Omron CX-Programmer project NewProject (CX-Programmer 9.73)

# PLC NewPLC1: CJ2M CPU11

## Global symbols (name address type ; comment)
D0.00 BOOL  ; Eixo X
D100 CHANNEL  ; Paletes Completas
D1000.00 BOOL  ; Sensor_P
D1000.01 BOOL  ; Sensor_M
D1000.02 BOOL  ; Sensor_G
D1000.03 BOOL  ; TI_P
D1000.04 BOOL  ; TI_M
D1000.05 BOOL  ; TI_G
D1000.06 BOOL  ; TF_P
D1000.07 BOOL  ; TF_M
D1000.08 BOOL  ; TF_G
D1000.09 BOOL  ; START
D1000.10 BOOL  ; STOP
D1000.11 BOOL  ; SensorPI
D1000.12 BOOL  ; Pick_Enable
D1000.13 BOOL  ; SensorPF
D1000.14 BOOL  ; C Limit
D1001.00 BOOL  ; Sensor_Palete
D1001.01 BOOL  ; Manual
D1001.02 BOOL  ; Auto
D1001.03 BOOL  ; Emergencia
D1001.04 BOOL  ; RESET
D101 CHANNEL  ; Cx Pequenas
D102 CHANNEL  ; Cx Médias
D103 CHANNEL  ; Cx Grandes
D104 CHANNEL  ; Eixo X Pick&Place
D104.00 BOOL  ; SPX
D105 CHANNEL  ; Eixo Y Pick&Place
D105.00 BOOL  ; SPY
D106 CHANNEL  ; Eixo Z Pick&Place
D106.00 BOOL  ; SPZ
D1.00 BOOL  ; Eixo Y
D2000.00 BOOL  ; TI
D2000.01 BOOL  ; Frente
D2000.02 BOOL  ; Esquerda
D2000.03 BOOL  ; Direita
D2000.04 BOOL  ; T_M
D2000.05 BOOL  ; T_P
D2000.06 BOOL  ; T_G
D2000.12 BOOL  ; GRAB
D2000.13 BOOL  ; Start_Light
D2000.14 BOOL  ; Stop_Light
D2001.01 BOOL  ; Remove_PaleteM
D2001.02 BOOL  ; Remove_PaleteP
D2001.03 BOOL  ; Remove_PaleteFull
D2001.04 BOOL  ; Atras
D2001.05 BOOL  ; Reset_Light
D2001.06 BOOL  ; Remove_PaleteG
D2001.07 BOOL  ; T_Palete
D2001.08 BOOL  ; Palete_Spawn
D2001.09 BOOL  ; Palete_Receive
D2001.10 BOOL  ; 90_ROT
D200.00 BOOL  ; E0- Sistema desligado
D200.01 BOOL  ; E1 - Sistema ligado
D200.02 BOOL  ; E2 - Decisão
D200.03 BOOL  ; E3 - Mover caixa pequena
D200.04 BOOL  ; E4 - Mover caixa média
D200.05 BOOL  ; E5 - Mover caixa grande
D200.06 BOOL  ; E6 - Palete Pronta
D200.07 BOOL  ; E7 - Braço elevado
D200.08 BOOL  ; E8 - X,Y Cx Pequena
D200.09 BOOL  ; E9 - X,Y Cx Média
D200.10 BOOL  ; E10 - X,Y Cx Grande
D200.11 BOOL  ; E11 - Pegar Cx Pequena
D200.12 BOOL  ; E12 - Pegar Cx Média
D200.13 BOOL  ; E13 - Pegar Cx Grande
D200.14 BOOL  ; E14 - Caixa recolhida
D200.15 BOOL  ; E15 - Palete Cx Pequena
D201.00 BOOL  ; E16 - Palete Cx Pequena x2
D201.01 BOOL  ; E17 - Palete Cx Média
D201.02 BOOL  ; E18 - Palete Cx Grande
D201.03 BOOL  ; E19.0 - Drop Caixa pequena
D201.04 BOOL  ; E20 - Drop Caixa grande
D201.05 BOOL  ; E21 - Caixa colocada
D201.06 BOOL  ; E22 - Palete Pronta
D201.07 BOOL  ; E23 - Recolher Palete
D201.08 BOOL  ; E19.1 - Drop Caixa pequena x2
D201.09 BOOL  ; E19.2 - Drop Caixa média
D2.00 BOOL  ; Eixo Z
D300.00 BOOL  ; ON
D300.01 BOOL  ; MP
D300.02 BOOL  ; MM
D300.03 BOOL  ; MG
D300.04 BOOL  ; PickInicio
D300.05 BOOL  ; Remove_PaleteG ON
D300.07 BOOL  ; PickPequena
D300.08 BOOL  ; PickMedia
D300.09 BOOL  ; PickGrande
D300.10 BOOL  ; Emergencia_ON
D300.11 BOOL  ; Auto_ON
D302.00 BOOL  ; Y>=3.69
D302.01 BOOL  ; Y<=371
D302.02 BOOL  ; Z>=7.69
D302.03 BOOL  ; Z<=7.71
D302.04 BOOL  ; Z>=5.29
D302.05 BOOL  ; Z<=5.31
D302.06 BOOL  ; Y>=2.59
D302.07 BOOL  ; Z<=2.61
D302.08 BOOL  ; Y>=1.29
D302.09 BOOL  ; Y<=1.31
D303.00 BOOL  ; Z=0
D303.01 BOOL  ; Y=3.7
D303.02 BOOL  ; Y=10
D303.03 BOOL  ; Z=7.7
D303.04 BOOL  ; Z=5.3
D303.05 BOOL  ; Y=2.6
D303.06 BOOL  ; Y=1.3
D303.07 BOOL  ; Y=0
D303.08 BOOL  ; Z=10
D304.00 BOOL  ; Move Cx_Pequena
D304.01 BOOL  ; Move Cx_Media
D304.02 BOOL  ; Move Cx_Grande
D304.03 BOOL  ; Pick Cx_Pequena
D304.04 BOOL  ; Drop Cx_Pequena1
D304.05 BOOL  ; Drop Cx_Pequena2
D304.06 BOOL  ; Pick Cx_Media
D304.07 BOOL  ; Drop Cx_Media
D304.08 BOOL  ; Pick Cx_Grande
D304.09 BOOL  ; Drop Cx_Grande
D304.10 BOOL  ; Move_Decisao
D304.11 BOOL  ; Tapete_Final
D304.12 BOOL  ; System_ON
D304.13 BOOL  ; Decisao_Ready
D304.14 BOOL  ; Control_Emergencia
D304.15 BOOL  ; Control_Auto
T0002 BOOL  ; Timer_MoveDecisao

## Program NewProgram1 (cyclic task 0)

### Section ACOES

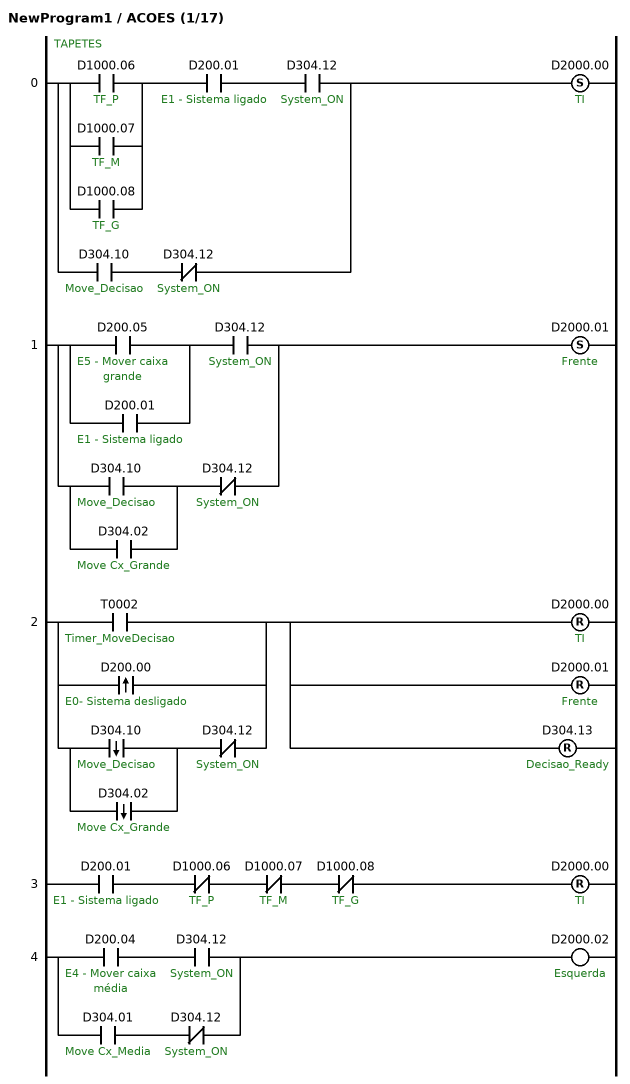
; rung 0: TAPETES
LD D1000.06  ; TF_P
OR D1000.07  ; TF_M
OR D1000.08  ; TF_G
AND D200.01  ; E1 - Sistema ligado
AND D304.12  ; System_ON
LD D304.10  ; Move_Decisao
ANDNOT D304.12  ; System_ON
ORLD
SET D2000.00  ; TI
; rung 1
LD D200.05  ; E5 - Mover caixa grande
OR D200.01  ; E1 - Sistema ligado
AND D304.12  ; System_ON
LD D304.10  ; Move_Decisao
OR D304.02  ; Move Cx_Grande
ANDNOT D304.12  ; System_ON
ORLD
SET D2000.01  ; Frente
; rung 2
LD T0002  ; Timer_MoveDecisao
@OR D200.00  ; E0- Sistema desligado
%LD D304.10  ; Move_Decisao
%OR D304.02  ; Move Cx_Grande
ANDNOT D304.12  ; System_ON
ORLD
RSET D2000.00  ; TI
RSET D2000.01  ; Frente
RSET D304.13  ; Decisao_Ready
; rung 3
LD D200.01  ; E1 - Sistema ligado
ANDNOT D1000.06  ; TF_P
ANDNOT D1000.07  ; TF_M
ANDNOT D1000.08  ; TF_G
RSET D2000.00  ; TI
; rung 4
LD D200.04  ; E4 - Mover caixa média
AND D304.12  ; System_ON
LD D304.01  ; Move Cx_Media
ANDNOT D304.12  ; System_ON
ORLD
OUT D2000.02  ; Esquerda

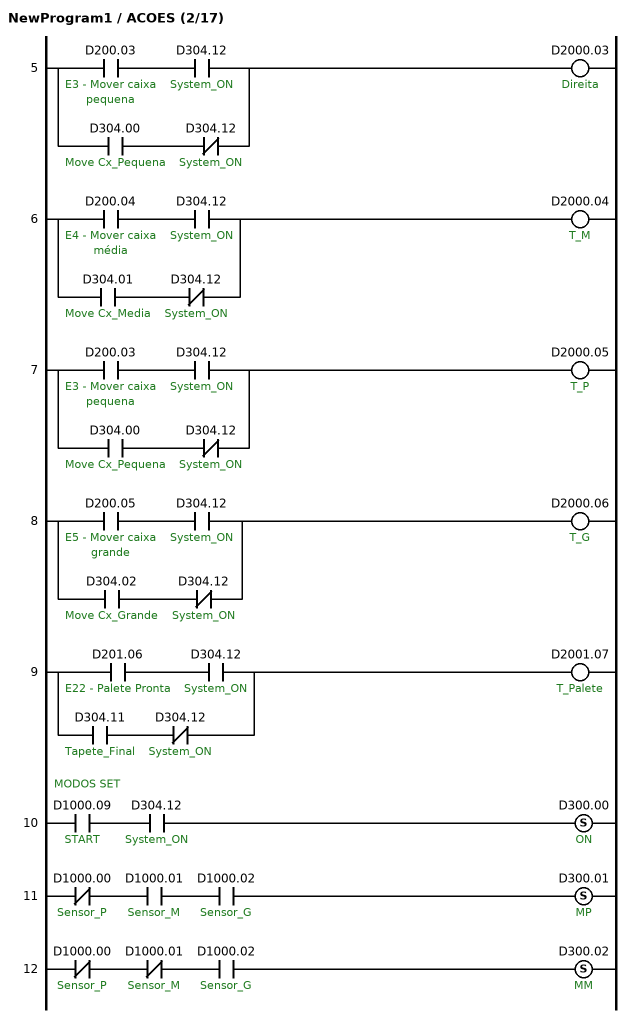
; rung 5
LD D200.03  ; E3 - Mover caixa pequena
AND D304.12  ; System_ON
LD D304.00  ; Move Cx_Pequena
ANDNOT D304.12  ; System_ON
ORLD
OUT D2000.03  ; Direita
; rung 6
LD D200.04  ; E4 - Mover caixa média
AND D304.12  ; System_ON
LD D304.01  ; Move Cx_Media
ANDNOT D304.12  ; System_ON
ORLD
OUT D2000.04  ; T_M
; rung 7
LD D200.03  ; E3 - Mover caixa pequena
AND D304.12  ; System_ON
LD D304.00  ; Move Cx_Pequena
ANDNOT D304.12  ; System_ON
ORLD
OUT D2000.05  ; T_P
; rung 8
LD D200.05  ; E5 - Mover caixa grande
AND D304.12  ; System_ON
LD D304.02  ; Move Cx_Grande
ANDNOT D304.12  ; System_ON
ORLD
OUT D2000.06  ; T_G
; rung 9
LD D201.06  ; E22 - Palete Pronta
AND D304.12  ; System_ON
LD D304.11  ; Tapete_Final
ANDNOT D304.12  ; System_ON
ORLD
OUT D2001.07  ; T_Palete
; rung 10: MODOS SET
LD D1000.09  ; START
AND D304.12  ; System_ON
SET D300.00  ; ON
; rung 11
LDNOT D1000.00  ; Sensor_P
AND D1000.01  ; Sensor_M
AND D1000.02  ; Sensor_G
SET D300.01  ; MP
; rung 12
LDNOT D1000.00  ; Sensor_P
ANDNOT D1000.01  ; Sensor_M
AND D1000.02  ; Sensor_G
SET D300.02  ; MM

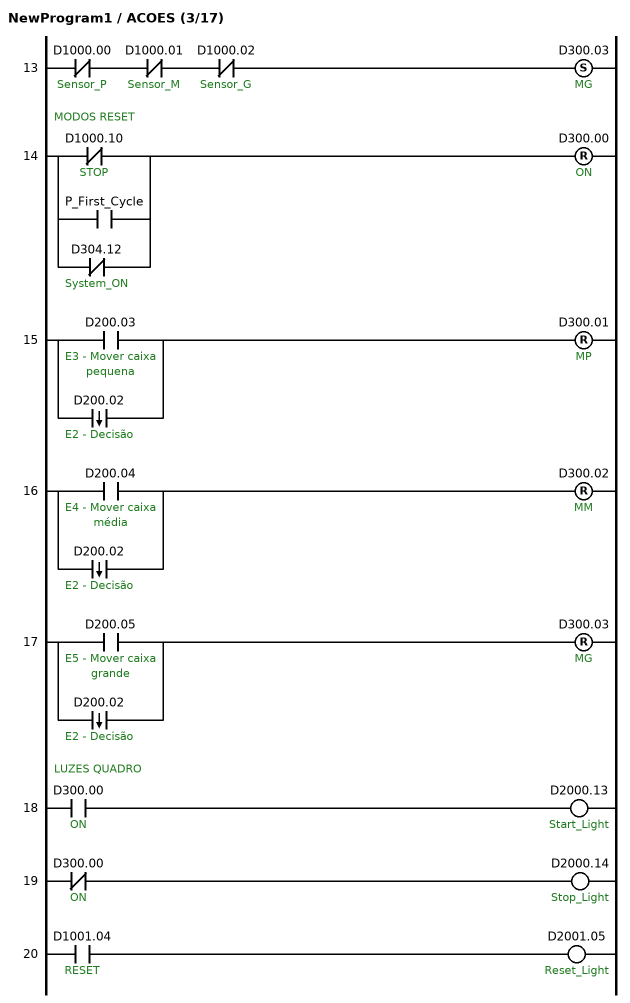
; rung 13
LDNOT D1000.00  ; Sensor_P
ANDNOT D1000.01  ; Sensor_M
ANDNOT D1000.02  ; Sensor_G
SET D300.03  ; MG
; rung 14: MODOS RESET
LDNOT D1000.10  ; STOP
OR P_First_Cycle
ORNOT D304.12  ; System_ON
RSET D300.00  ; ON
; rung 15
LD D200.03  ; E3 - Mover caixa pequena
%OR D200.02  ; E2 - Decisão
RSET D300.01  ; MP
; rung 16
LD D200.04  ; E4 - Mover caixa média
%OR D200.02  ; E2 - Decisão
RSET D300.02  ; MM
; rung 17
LD D200.05  ; E5 - Mover caixa grande
%OR D200.02  ; E2 - Decisão
RSET D300.03  ; MG
; rung 18: LUZES QUADRO
LD D300.00  ; ON
OUT D2000.13  ; Start_Light
; rung 19
LDNOT D300.00  ; ON
OUT D2000.14  ; Stop_Light
; rung 20
LD D1001.04  ; RESET
OUT D2001.05  ; Reset_Light

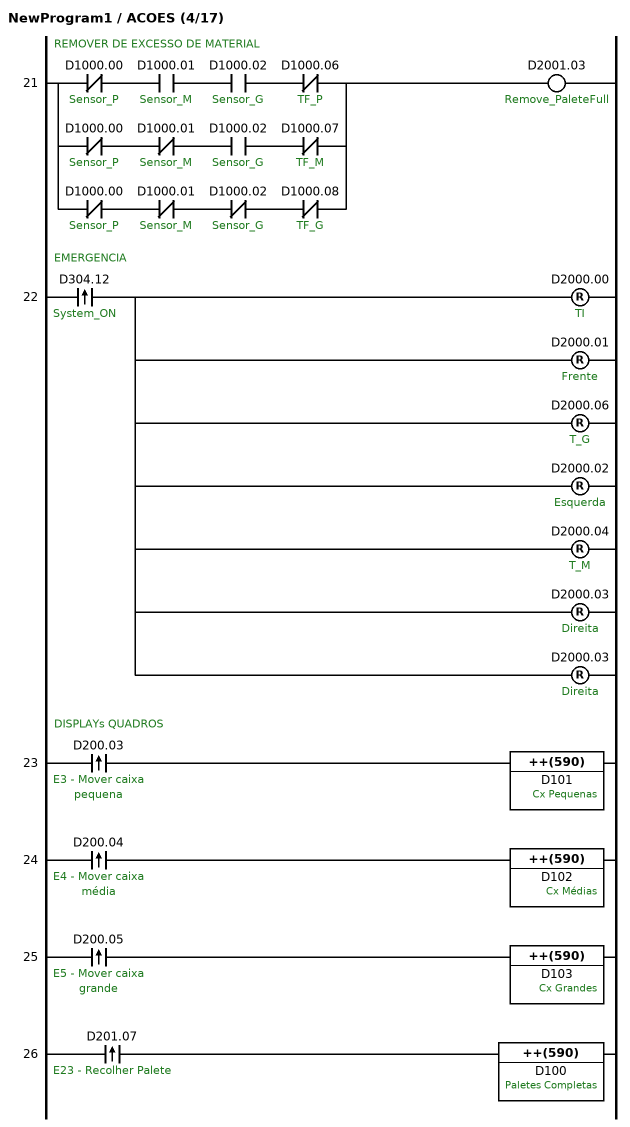
; rung 21: REMOVER DE EXCESSO DE MATERIAL
LDNOT D1000.00  ; Sensor_P
AND D1000.01  ; Sensor_M
AND D1000.02  ; Sensor_G
ANDNOT D1000.06  ; TF_P
LDNOT D1000.00  ; Sensor_P
ANDNOT D1000.01  ; Sensor_M
AND D1000.02  ; Sensor_G
ANDNOT D1000.07  ; TF_M
ORLD
LDNOT D1000.00  ; Sensor_P
ANDNOT D1000.01  ; Sensor_M
ANDNOT D1000.02  ; Sensor_G
ANDNOT D1000.08  ; TF_G
ORLD
OUT D2001.03  ; Remove_PaleteFull
; rung 22: EMERGENCIA
@LD D304.12  ; System_ON
RSET D2000.00  ; TI
RSET D2000.01  ; Frente
RSET D2000.06  ; T_G
RSET D2000.02  ; Esquerda
RSET D2000.04  ; T_M
RSET D2000.03  ; Direita
RSET D2000.03  ; Direita
; rung 23: DISPLAYs QUADROS
@LD D200.03  ; E3 - Mover caixa pequena
++(590) D101  ; Cx Pequenas
; rung 24
@LD D200.04  ; E4 - Mover caixa média
++(590) D102  ; Cx Médias
; rung 25
@LD D200.05  ; E5 - Mover caixa grande
++(590) D103  ; Cx Grandes
; rung 26
@LD D201.07  ; E23 - Recolher Palete
++(590) D100  ; Paletes Completas

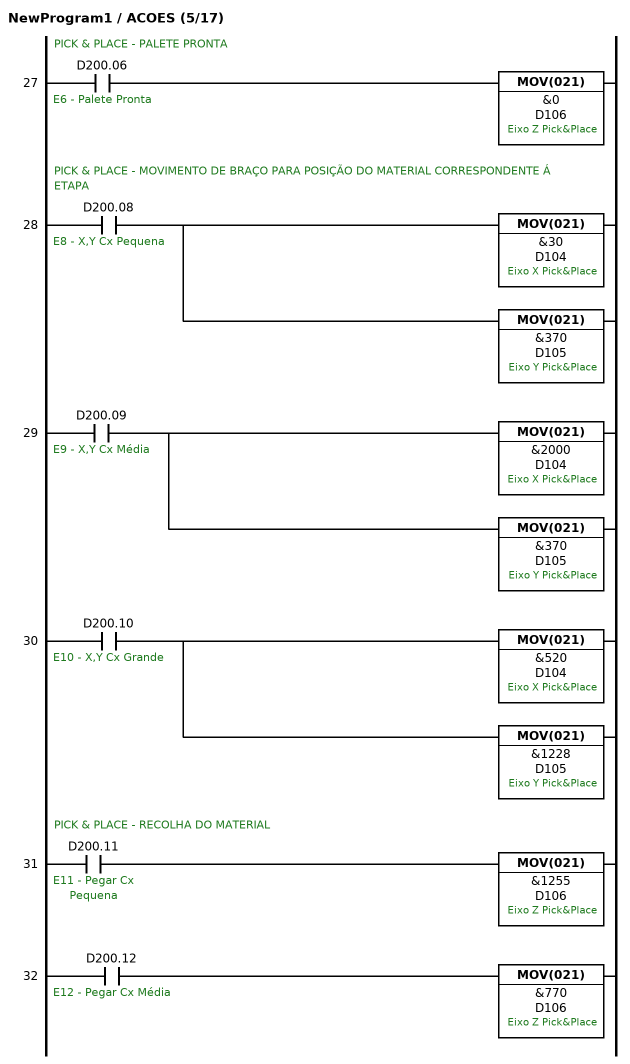
; rung 27: PICK & PLACE - PALETE PRONTA
LD D200.06  ; E6 - Palete Pronta
MOV(021) &0 D106  ; Eixo Z Pick&Place
; rung 28: PICK & PLACE - MOVIMENTO DE BRAÇO PARA POSIÇÃO DO MATERIAL CORRESPONDENTE Á ETAPA
LD D200.08  ; E8 - X,Y Cx Pequena
MOV(021) &30 D104  ; Eixo X Pick&Place
MOV(021) &370 D105  ; Eixo Y Pick&Place
; rung 29
LD D200.09  ; E9 - X,Y Cx Média
MOV(021) &2000 D104  ; Eixo X Pick&Place
MOV(021) &370 D105  ; Eixo Y Pick&Place
; rung 30
LD D200.10  ; E10 - X,Y Cx Grande
MOV(021) &520 D104  ; Eixo X Pick&Place
MOV(021) &1228 D105  ; Eixo Y Pick&Place
; rung 31: PICK & PLACE - RECOLHA DO MATERIAL
LD D200.11  ; E11 - Pegar Cx Pequena
MOV(021) &1255 D106  ; Eixo Z Pick&Place
; rung 32
LD D200.12  ; E12 - Pegar Cx Média
MOV(021) &770 D106  ; Eixo Z Pick&Place

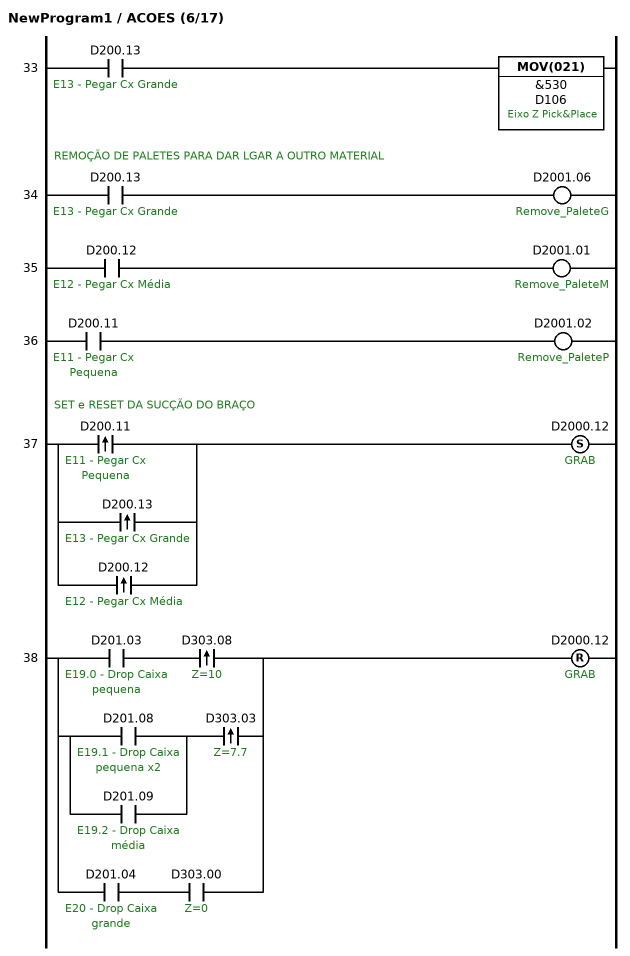
; rung 33
LD D200.13  ; E13 - Pegar Cx Grande
MOV(021) &530 D106  ; Eixo Z Pick&Place
; rung 34: REMOÇÃO DE PALETES PARA DAR LGAR A OUTRO MATERIAL
LD D200.13  ; E13 - Pegar Cx Grande
OUT D2001.06  ; Remove_PaleteG
; rung 35
LD D200.12  ; E12 - Pegar Cx Média
OUT D2001.01  ; Remove_PaleteM
; rung 36
LD D200.11  ; E11 - Pegar Cx Pequena
OUT D2001.02  ; Remove_PaleteP
; rung 37: SET e RESET DA SUCÇÃO DO BRAÇO
@LD D200.11  ; E11 - Pegar Cx Pequena
@OR D200.13  ; E13 - Pegar Cx Grande
@OR D200.12  ; E12 - Pegar Cx Média
SET D2000.12  ; GRAB
; rung 38
LD D201.03  ; E19.0 - Drop Caixa pequena
@AND D303.08  ; Z=10
LD D201.08  ; E19.1 - Drop Caixa pequena x2
OR D201.09  ; E19.2 - Drop Caixa média
@AND D303.03  ; Z=7.7
ORLD
LD D201.04  ; E20 - Drop Caixa grande
AND D303.00  ; Z=0
ORLD
RSET D2000.12  ; GRAB

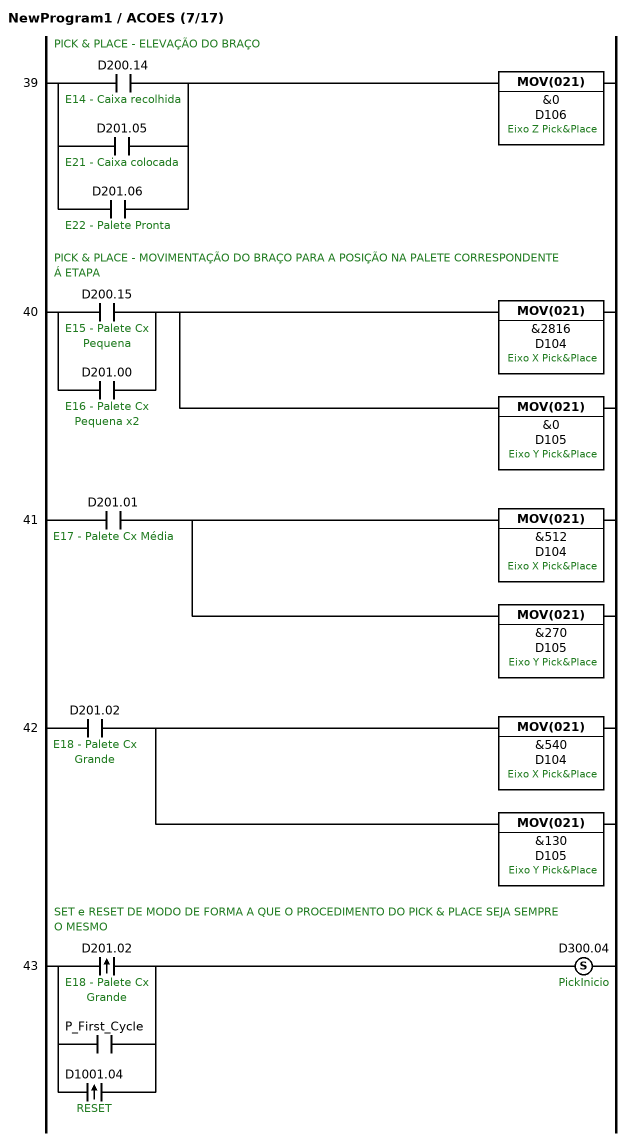
; rung 39: PICK & PLACE - ELEVAÇÃO DO BRAÇO
LD D200.14  ; E14 - Caixa recolhida
OR D201.05  ; E21 - Caixa colocada
OR D201.06  ; E22 - Palete Pronta
MOV(021) &0 D106  ; Eixo Z Pick&Place
; rung 40: PICK & PLACE - MOVIMENTAÇÃO DO BRAÇO PARA A POSIÇÃO NA PALETE CORRESPONDENTE Á ETAPA
LD D200.15  ; E15 - Palete Cx Pequena
OR D201.00  ; E16 - Palete Cx Pequena x2
MOV(021) &2816 D104  ; Eixo X Pick&Place
MOV(021) &0 D105  ; Eixo Y Pick&Place
; rung 41
LD D201.01  ; E17 - Palete Cx Média
MOV(021) &512 D104  ; Eixo X Pick&Place
MOV(021) &270 D105  ; Eixo Y Pick&Place
; rung 42
LD D201.02  ; E18 - Palete Cx Grande
MOV(021) &540 D104  ; Eixo X Pick&Place
MOV(021) &130 D105  ; Eixo Y Pick&Place
; rung 43: SET e RESET DE MODO DE FORMA A QUE O PROCEDIMENTO DO PICK & PLACE SEJA SEMPRE O MESMO
@LD D201.02  ; E18 - Palete Cx Grande
OR P_First_Cycle
@OR D1001.04  ; RESET
SET D300.04  ; PickInicio

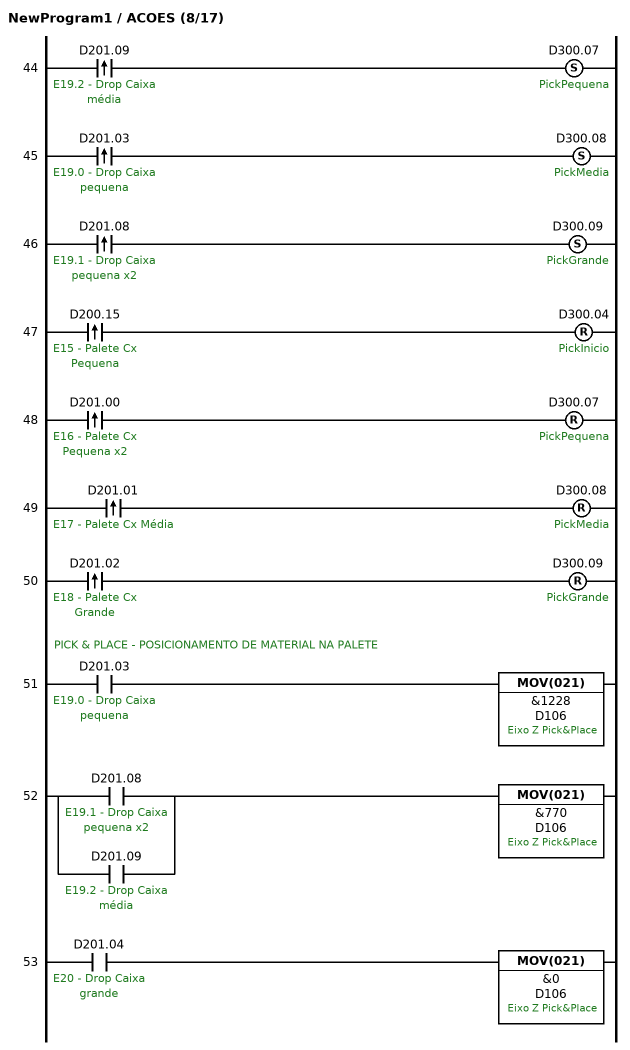
; rung 44
@LD D201.09  ; E19.2 - Drop Caixa média
SET D300.07  ; PickPequena
; rung 45
@LD D201.03  ; E19.0 - Drop Caixa pequena
SET D300.08  ; PickMedia
; rung 46
@LD D201.08  ; E19.1 - Drop Caixa pequena x2
SET D300.09  ; PickGrande
; rung 47
@LD D200.15  ; E15 - Palete Cx Pequena
RSET D300.04  ; PickInicio
; rung 48
@LD D201.00  ; E16 - Palete Cx Pequena x2
RSET D300.07  ; PickPequena
; rung 49
@LD D201.01  ; E17 - Palete Cx Média
RSET D300.08  ; PickMedia
; rung 50
@LD D201.02  ; E18 - Palete Cx Grande
RSET D300.09  ; PickGrande
; rung 51: PICK & PLACE - POSICIONAMENTO DE MATERIAL NA PALETE
LD D201.03  ; E19.0 - Drop Caixa pequena
MOV(021) &1228 D106  ; Eixo Z Pick&Place
; rung 52
LD D201.08  ; E19.1 - Drop Caixa pequena x2
OR D201.09  ; E19.2 - Drop Caixa média
MOV(021) &770 D106  ; Eixo Z Pick&Place
; rung 53
LD D201.04  ; E20 - Drop Caixa grande
MOV(021) &0 D106  ; Eixo Z Pick&Place

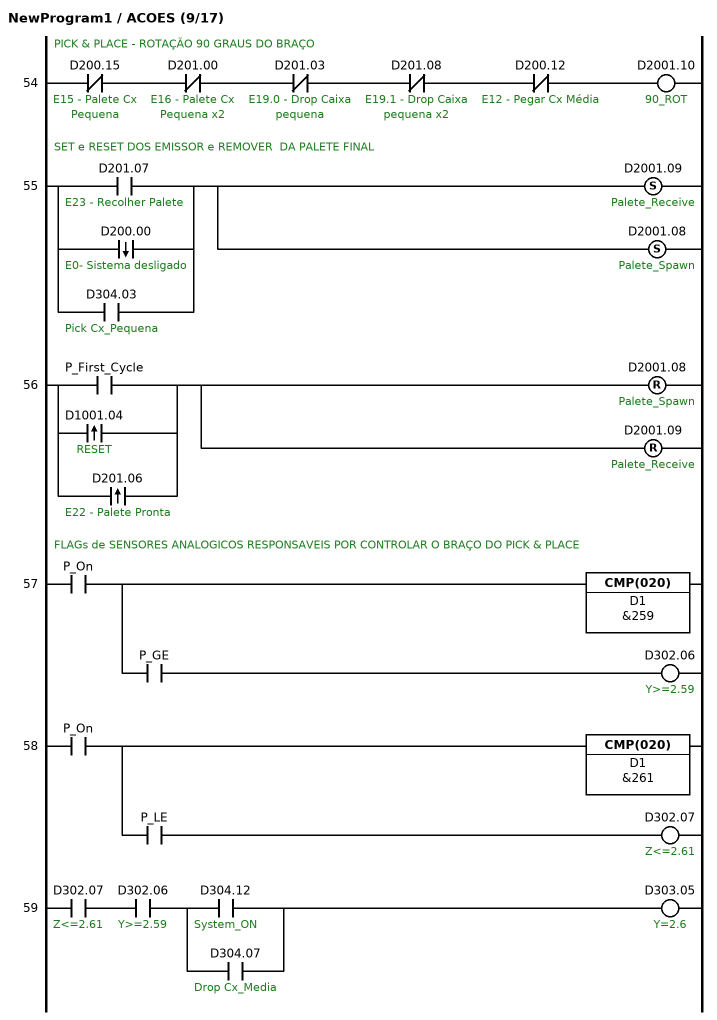
; rung 54: PICK & PLACE - ROTAÇÃO 90 GRAUS DO BRAÇO
LDNOT D200.15  ; E15 - Palete Cx Pequena
ANDNOT D201.00  ; E16 - Palete Cx Pequena x2
ANDNOT D201.03  ; E19.0 - Drop Caixa pequena
ANDNOT D201.08  ; E19.1 - Drop Caixa pequena x2
ANDNOT D200.12  ; E12 - Pegar Cx Média
OUT D2001.10  ; 90_ROT
; rung 55: SET e RESET DOS EMISSOR e REMOVER  DA PALETE FINAL
LD D201.07  ; E23 - Recolher Palete
%OR D200.00  ; E0- Sistema desligado
OR D304.03  ; Pick Cx_Pequena
SET D2001.09  ; Palete_Receive
SET D2001.08  ; Palete_Spawn
; rung 56
LD P_First_Cycle
@OR D1001.04  ; RESET
@OR D201.06  ; E22 - Palete Pronta
RSET D2001.08  ; Palete_Spawn
RSET D2001.09  ; Palete_Receive
; rung 57: FLAGs de SENSORES ANALOGICOS RESPONSAVEIS POR CONTROLAR O BRAÇO DO PICK & PLACE
LD P_On
CMP(020) D1 &259
AND P_GE
OUT D302.06  ; Y>=2.59
; rung 58
LD P_On
CMP(020) D1 &261
AND P_LE
OUT D302.07  ; Z<=2.61
; rung 59
LD D302.07  ; Z<=2.61
AND D302.06  ; Y>=2.59
LD D304.12  ; System_ON
OR D304.07  ; Drop Cx_Media
ANDLD
OUT D303.05  ; Y=2.6

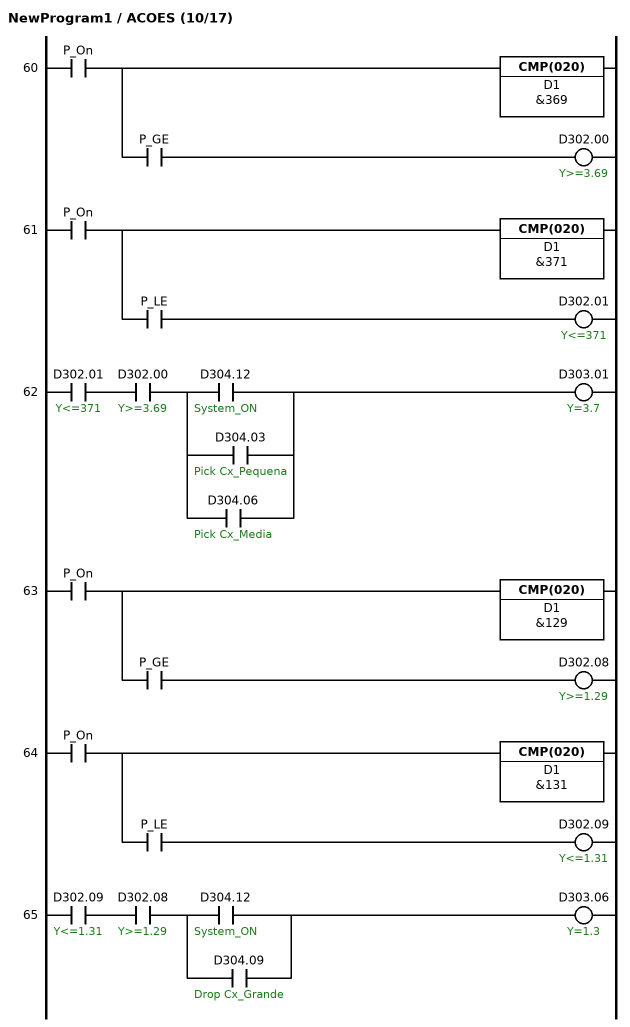
; rung 60
LD P_On
CMP(020) D1 &369
AND P_GE
OUT D302.00  ; Y>=3.69
; rung 61
LD P_On
CMP(020) D1 &371
AND P_LE
OUT D302.01  ; Y<=371
; rung 62
LD D302.01  ; Y<=371
AND D302.00  ; Y>=3.69
LD D304.12  ; System_ON
OR D304.03  ; Pick Cx_Pequena
OR D304.06  ; Pick Cx_Media
ANDLD
OUT D303.01  ; Y=3.7
; rung 63
LD P_On
CMP(020) D1 &129
AND P_GE
OUT D302.08  ; Y>=1.29
; rung 64
LD P_On
CMP(020) D1 &131
AND P_LE
OUT D302.09  ; Y<=1.31
; rung 65
LD D302.09  ; Y<=1.31
AND D302.08  ; Y>=1.29
LD D304.12  ; System_ON
OR D304.09  ; Drop Cx_Grande
ANDLD
OUT D303.06  ; Y=1.3

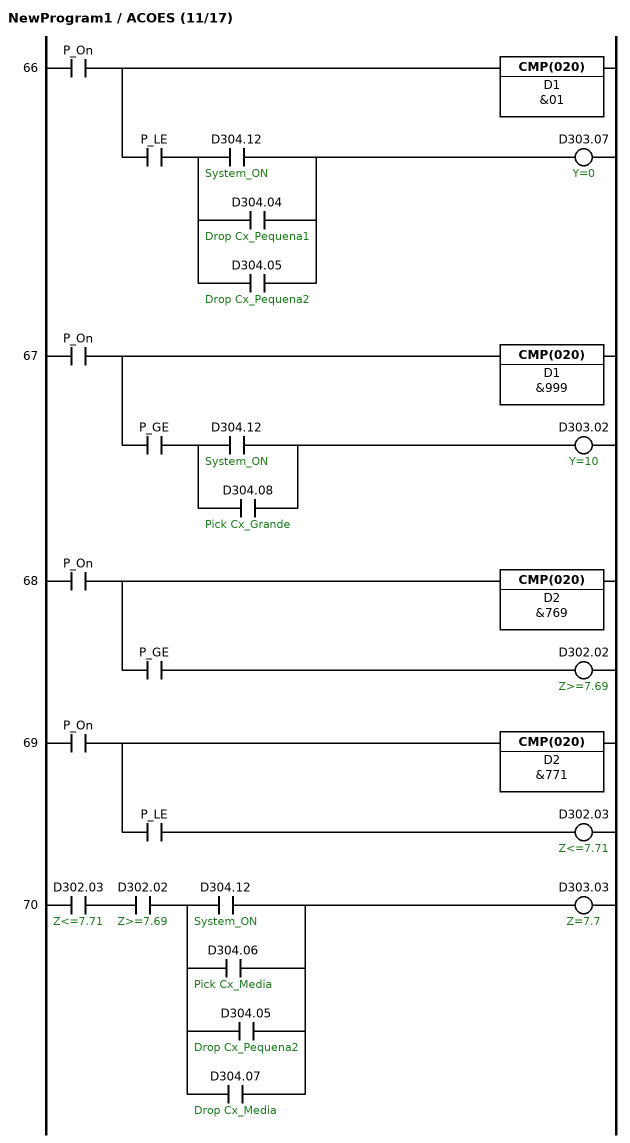
; rung 66
LD P_On
CMP(020) D1 &01
AND P_LE
LD D304.12  ; System_ON
OR D304.04  ; Drop Cx_Pequena1
OR D304.05  ; Drop Cx_Pequena2
ANDLD
OUT D303.07  ; Y=0
; rung 67
LD P_On
CMP(020) D1 &999
AND P_GE
LD D304.12  ; System_ON
OR D304.08  ; Pick Cx_Grande
ANDLD
OUT D303.02  ; Y=10
; rung 68
LD P_On
CMP(020) D2 &769
AND P_GE
OUT D302.02  ; Z>=7.69
; rung 69
LD P_On
CMP(020) D2 &771
AND P_LE
OUT D302.03  ; Z<=7.71
; rung 70
LD D302.03  ; Z<=7.71
AND D302.02  ; Z>=7.69
LD D304.12  ; System_ON
OR D304.06  ; Pick Cx_Media
OR D304.05  ; Drop Cx_Pequena2
OR D304.07  ; Drop Cx_Media
ANDLD
OUT D303.03  ; Z=7.7

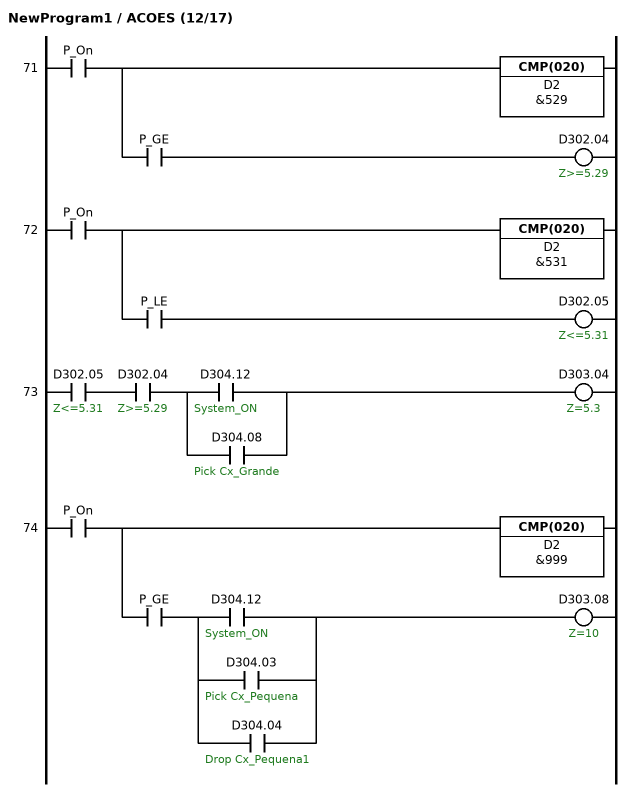
; rung 71
LD P_On
CMP(020) D2 &529
AND P_GE
OUT D302.04  ; Z>=5.29
; rung 72
LD P_On
CMP(020) D2 &531
AND P_LE
OUT D302.05  ; Z<=5.31
; rung 73
LD D302.05  ; Z<=5.31
AND D302.04  ; Z>=5.29
LD D304.12  ; System_ON
OR D304.08  ; Pick Cx_Grande
ANDLD
OUT D303.04  ; Z=5.3
; rung 74
LD P_On
CMP(020) D2 &999
AND P_GE
LD D304.12  ; System_ON
OR D304.03  ; Pick Cx_Pequena
OR D304.04  ; Drop Cx_Pequena1
ANDLD
OUT D303.08  ; Z=10

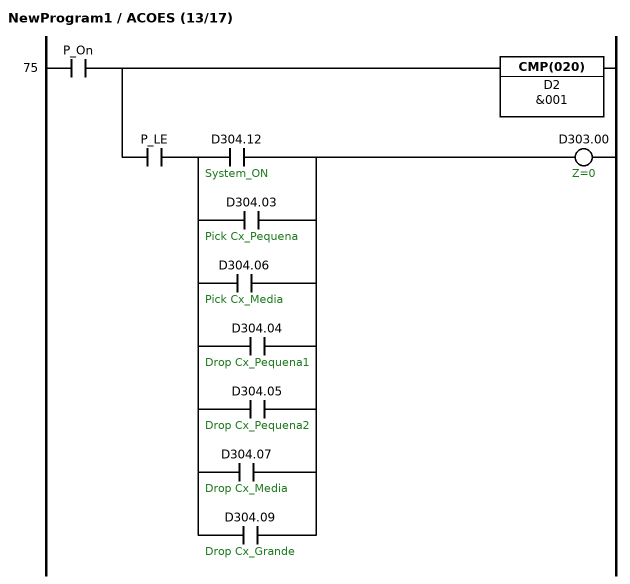
; rung 75
LD P_On
CMP(020) D2 &001
AND P_LE
LD D304.12  ; System_ON
OR D304.03  ; Pick Cx_Pequena
OR D304.06  ; Pick Cx_Media
OR D304.04  ; Drop Cx_Pequena1
OR D304.05  ; Drop Cx_Pequena2
OR D304.07  ; Drop Cx_Media
OR D304.09  ; Drop Cx_Grande
ANDLD
OUT D303.00  ; Z=0

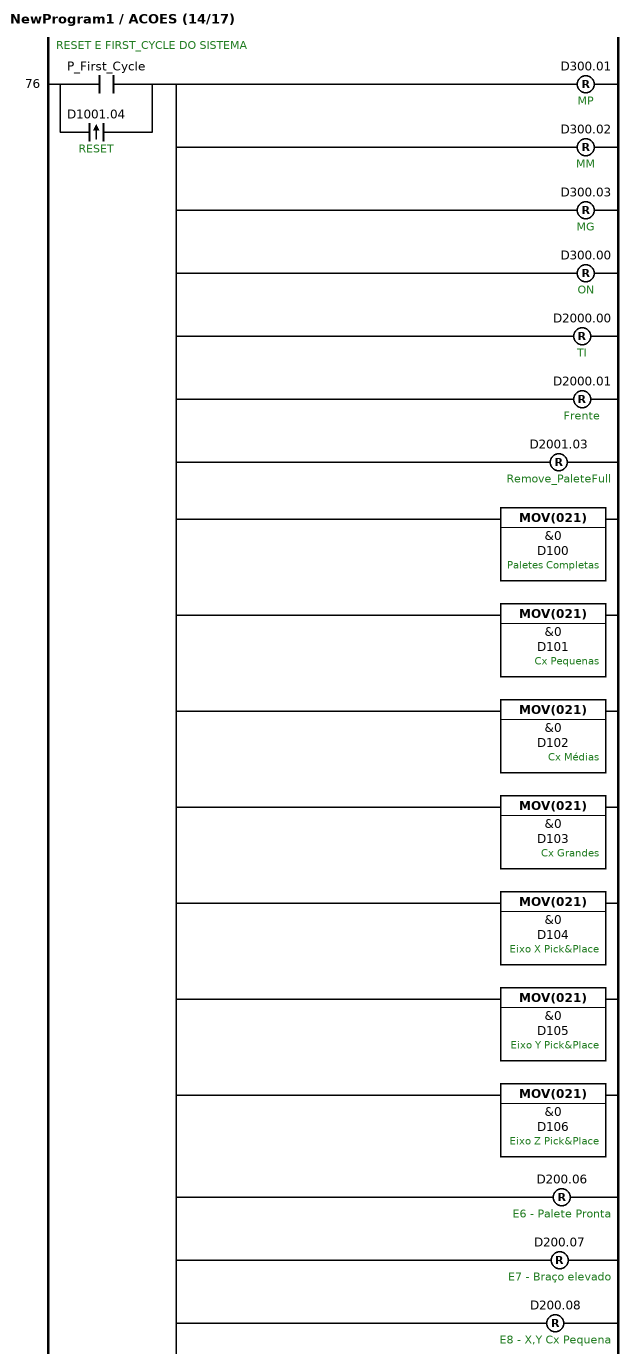

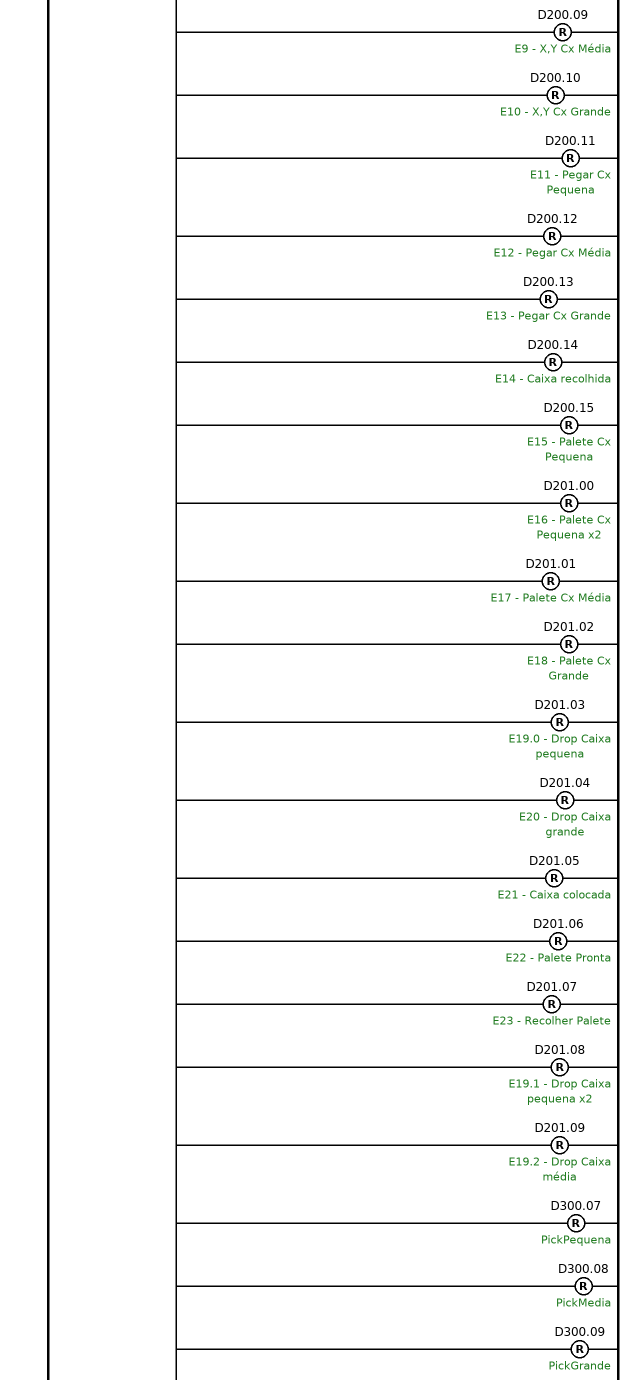

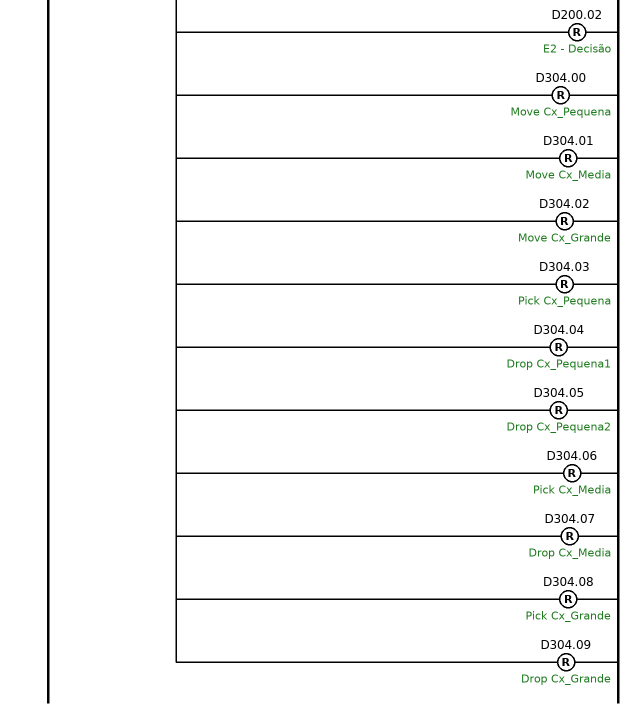
; rung 76: RESET E FIRST_CYCLE DO SISTEMA
LD P_First_Cycle
@OR D1001.04  ; RESET
RSET D300.01  ; MP
RSET D300.02  ; MM
RSET D300.03  ; MG
RSET D300.00  ; ON
RSET D2000.00  ; TI
RSET D2000.01  ; Frente
RSET D2001.03  ; Remove_PaleteFull
MOV(021) &0 D100  ; Paletes Completas
MOV(021) &0 D101  ; Cx Pequenas
MOV(021) &0 D102  ; Cx Médias
MOV(021) &0 D103  ; Cx Grandes
MOV(021) &0 D104  ; Eixo X Pick&Place
MOV(021) &0 D105  ; Eixo Y Pick&Place
MOV(021) &0 D106  ; Eixo Z Pick&Place
RSET D200.06  ; E6 - Palete Pronta
RSET D200.07  ; E7 - Braço elevado
RSET D200.08  ; E8 - X,Y Cx Pequena
RSET D200.09  ; E9 - X,Y Cx Média
RSET D200.10  ; E10 - X,Y Cx Grande
RSET D200.11  ; E11 - Pegar Cx Pequena
RSET D200.12  ; E12 - Pegar Cx Média
RSET D200.13  ; E13 - Pegar Cx Grande
RSET D200.14  ; E14 - Caixa recolhida
RSET D200.15  ; E15 - Palete Cx Pequena
RSET D201.00  ; E16 - Palete Cx Pequena x2
RSET D201.01  ; E17 - Palete Cx Média
RSET D201.02  ; E18 - Palete Cx Grande
RSET D201.03  ; E19.0 - Drop Caixa pequena
RSET D201.04  ; E20 - Drop Caixa grande
RSET D201.05  ; E21 - Caixa colocada
RSET D201.06  ; E22 - Palete Pronta
RSET D201.07  ; E23 - Recolher Palete
RSET D201.08  ; E19.1 - Drop Caixa pequena x2
RSET D201.09  ; E19.2 - Drop Caixa média
RSET D300.07  ; PickPequena
RSET D300.08  ; PickMedia
RSET D300.09  ; PickGrande
RSET D200.02  ; E2 - Decisão
RSET D304.00  ; Move Cx_Pequena
RSET D304.01  ; Move Cx_Media
RSET D304.02  ; Move Cx_Grande
RSET D304.03  ; Pick Cx_Pequena
RSET D304.04  ; Drop Cx_Pequena1
RSET D304.05  ; Drop Cx_Pequena2
RSET D304.06  ; Pick Cx_Media
RSET D304.07  ; Drop Cx_Media
RSET D304.08  ; Pick Cx_Grande
RSET D304.09  ; Drop Cx_Grande

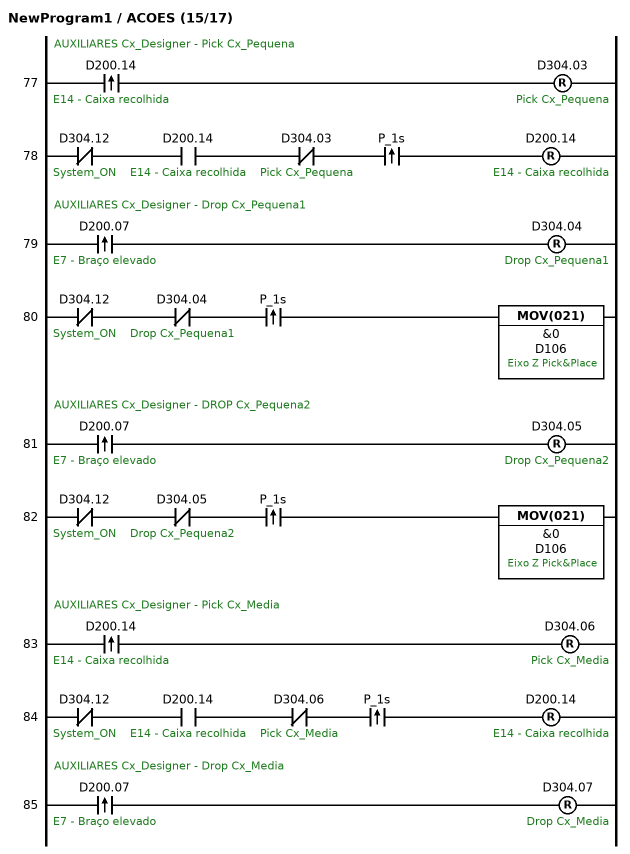
; rung 77: AUXILIARES Cx_Designer - Pick Cx_Pequena
@LD D200.14  ; E14 - Caixa recolhida
RSET D304.03  ; Pick Cx_Pequena
; rung 78
LDNOT D304.12  ; System_ON
AND D200.14  ; E14 - Caixa recolhida
ANDNOT D304.03  ; Pick Cx_Pequena
@AND P_1s
RSET D200.14  ; E14 - Caixa recolhida
; rung 79: AUXILIARES Cx_Designer - Drop Cx_Pequena1
@LD D200.07  ; E7 - Braço elevado
RSET D304.04  ; Drop Cx_Pequena1
; rung 80
LDNOT D304.12  ; System_ON
ANDNOT D304.04  ; Drop Cx_Pequena1
@AND P_1s
MOV(021) &0 D106  ; Eixo Z Pick&Place
; rung 81: AUXILIARES Cx_Designer - DROP Cx_Pequena2
@LD D200.07  ; E7 - Braço elevado
RSET D304.05  ; Drop Cx_Pequena2
; rung 82
LDNOT D304.12  ; System_ON
ANDNOT D304.05  ; Drop Cx_Pequena2
@AND P_1s
MOV(021) &0 D106  ; Eixo Z Pick&Place
; rung 83: AUXILIARES Cx_Designer - Pick Cx_Media
@LD D200.14  ; E14 - Caixa recolhida
RSET D304.06  ; Pick Cx_Media
; rung 84
LDNOT D304.12  ; System_ON
AND D200.14  ; E14 - Caixa recolhida
ANDNOT D304.06  ; Pick Cx_Media
@AND P_1s
RSET D200.14  ; E14 - Caixa recolhida
; rung 85: AUXILIARES Cx_Designer - Drop Cx_Media
@LD D200.07  ; E7 - Braço elevado
RSET D304.07  ; Drop Cx_Media

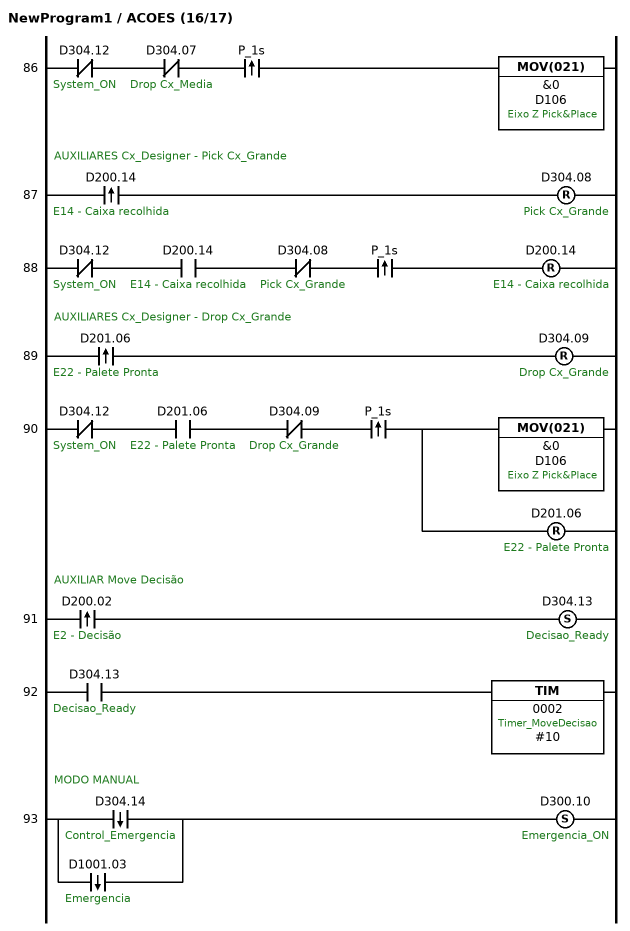
; rung 86
LDNOT D304.12  ; System_ON
ANDNOT D304.07  ; Drop Cx_Media
@AND P_1s
MOV(021) &0 D106  ; Eixo Z Pick&Place
; rung 87: AUXILIARES Cx_Designer - Pick Cx_Grande
@LD D200.14  ; E14 - Caixa recolhida
RSET D304.08  ; Pick Cx_Grande
; rung 88
LDNOT D304.12  ; System_ON
AND D200.14  ; E14 - Caixa recolhida
ANDNOT D304.08  ; Pick Cx_Grande
@AND P_1s
RSET D200.14  ; E14 - Caixa recolhida
; rung 89: AUXILIARES Cx_Designer - Drop Cx_Grande
@LD D201.06  ; E22 - Palete Pronta
RSET D304.09  ; Drop Cx_Grande
; rung 90
LDNOT D304.12  ; System_ON
AND D201.06  ; E22 - Palete Pronta
ANDNOT D304.09  ; Drop Cx_Grande
@AND P_1s
MOV(021) &0 D106  ; Eixo Z Pick&Place
RSET D201.06  ; E22 - Palete Pronta
; rung 91: AUXILIAR Move Decisão
@LD D200.02  ; E2 - Decisão
SET D304.13  ; Decisao_Ready
; rung 92
LD D304.13  ; Decisao_Ready
TIM 0002 #10  ; Timer_MoveDecisao
; rung 93: MODO MANUAL
%LD D304.14  ; Control_Emergencia
%OR D1001.03  ; Emergencia
SET D300.10  ; Emergencia_ON

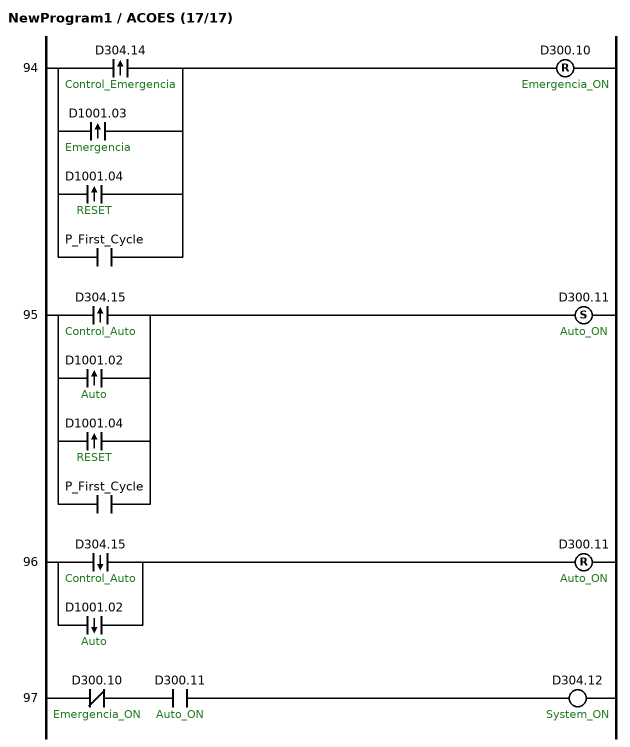
; rung 94
@LD D304.14  ; Control_Emergencia
@OR D1001.03  ; Emergencia
@OR D1001.04  ; RESET
OR P_First_Cycle
RSET D300.10  ; Emergencia_ON
; rung 95
@LD D304.15  ; Control_Auto
@OR D1001.02  ; Auto
@OR D1001.04  ; RESET
OR P_First_Cycle
SET D300.11  ; Auto_ON
; rung 96
%LD D304.15  ; Control_Auto
%OR D1001.02  ; Auto
RSET D300.11  ; Auto_ON
; rung 97
LDNOT D300.10  ; Emergencia_ON
AND D300.11  ; Auto_ON
OUT D304.12  ; System_ON

### Section ETAPAS

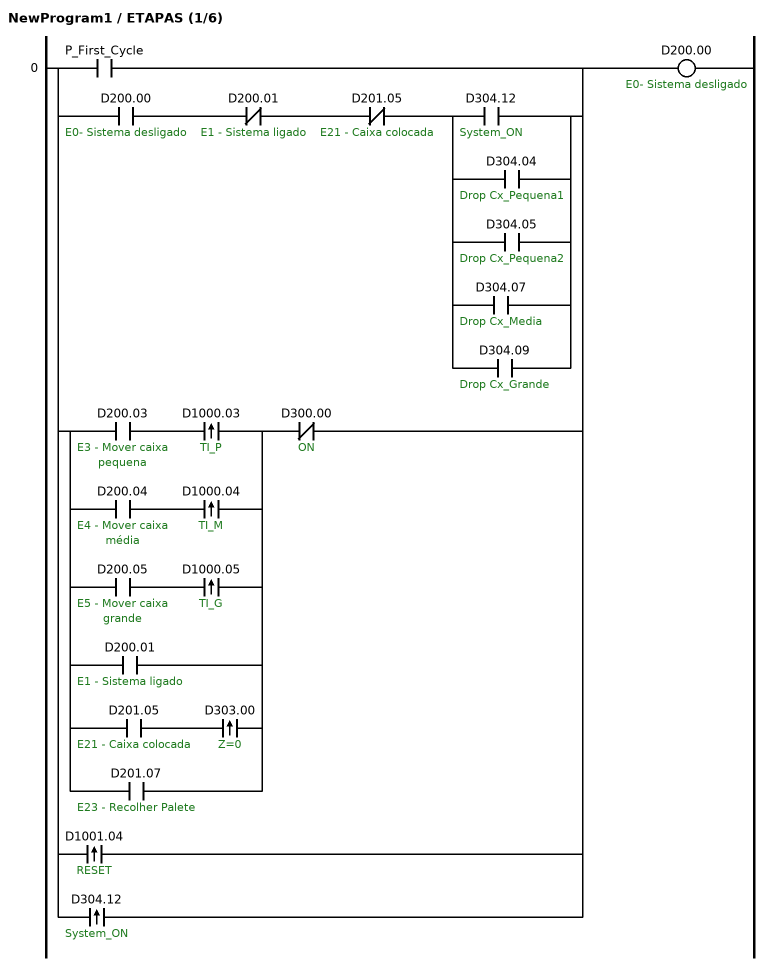
; rung 0
LD P_First_Cycle
LD D200.00  ; E0- Sistema desligado
ANDNOT D200.01  ; E1 - Sistema ligado
ANDNOT D201.05  ; E21 - Caixa colocada
LD D304.12  ; System_ON
OR D304.04  ; Drop Cx_Pequena1
OR D304.05  ; Drop Cx_Pequena2
OR D304.07  ; Drop Cx_Media
OR D304.09  ; Drop Cx_Grande
ANDLD
ORLD
LD D200.03  ; E3 - Mover caixa pequena
@AND D1000.03  ; TI_P
LD D200.04  ; E4 - Mover caixa média
@AND D1000.04  ; TI_M
ORLD
LD D200.05  ; E5 - Mover caixa grande
@AND D1000.05  ; TI_G
ORLD
OR D200.01  ; E1 - Sistema ligado
LD D201.05  ; E21 - Caixa colocada
@AND D303.00  ; Z=0
ORLD
OR D201.07  ; E23 - Recolher Palete
ANDNOT D300.00  ; ON
ORLD
@OR D1001.04  ; RESET
@OR D304.12  ; System_ON
OUT D200.00  ; E0- Sistema desligado

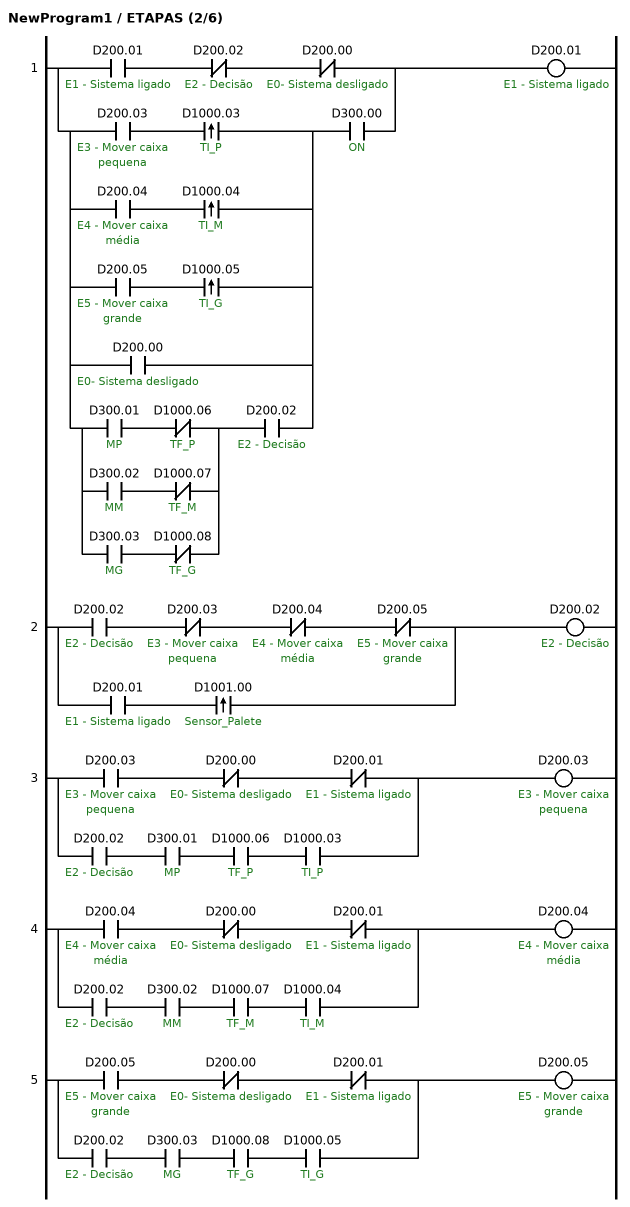
; rung 1
LD D200.01  ; E1 - Sistema ligado
ANDNOT D200.02  ; E2 - Decisão
ANDNOT D200.00  ; E0- Sistema desligado
LD D200.03  ; E3 - Mover caixa pequena
@AND D1000.03  ; TI_P
LD D200.04  ; E4 - Mover caixa média
@AND D1000.04  ; TI_M
ORLD
LD D200.05  ; E5 - Mover caixa grande
@AND D1000.05  ; TI_G
ORLD
OR D200.00  ; E0- Sistema desligado
LD D300.01  ; MP
ANDNOT D1000.06  ; TF_P
LD D300.02  ; MM
ANDNOT D1000.07  ; TF_M
ORLD
LD D300.03  ; MG
ANDNOT D1000.08  ; TF_G
ORLD
AND D200.02  ; E2 - Decisão
ORLD
AND D300.00  ; ON
ORLD
OUT D200.01  ; E1 - Sistema ligado
; rung 2
LD D200.02  ; E2 - Decisão
ANDNOT D200.03  ; E3 - Mover caixa pequena
ANDNOT D200.04  ; E4 - Mover caixa média
ANDNOT D200.05  ; E5 - Mover caixa grande
LD D200.01  ; E1 - Sistema ligado
@AND D1001.00  ; Sensor_Palete
ORLD
OUT D200.02  ; E2 - Decisão
; rung 3
LD D200.03  ; E3 - Mover caixa pequena
ANDNOT D200.00  ; E0- Sistema desligado
ANDNOT D200.01  ; E1 - Sistema ligado
LD D200.02  ; E2 - Decisão
AND D300.01  ; MP
AND D1000.06  ; TF_P
AND D1000.03  ; TI_P
ORLD
OUT D200.03  ; E3 - Mover caixa pequena
; rung 4
LD D200.04  ; E4 - Mover caixa média
ANDNOT D200.00  ; E0- Sistema desligado
ANDNOT D200.01  ; E1 - Sistema ligado
LD D200.02  ; E2 - Decisão
AND D300.02  ; MM
AND D1000.07  ; TF_M
AND D1000.04  ; TI_M
ORLD
OUT D200.04  ; E4 - Mover caixa média
; rung 5
LD D200.05  ; E5 - Mover caixa grande
ANDNOT D200.00  ; E0- Sistema desligado
ANDNOT D200.01  ; E1 - Sistema ligado
LD D200.02  ; E2 - Decisão
AND D300.03  ; MG
AND D1000.08  ; TF_G
AND D1000.05  ; TI_G
ORLD
OUT D200.05  ; E5 - Mover caixa grande

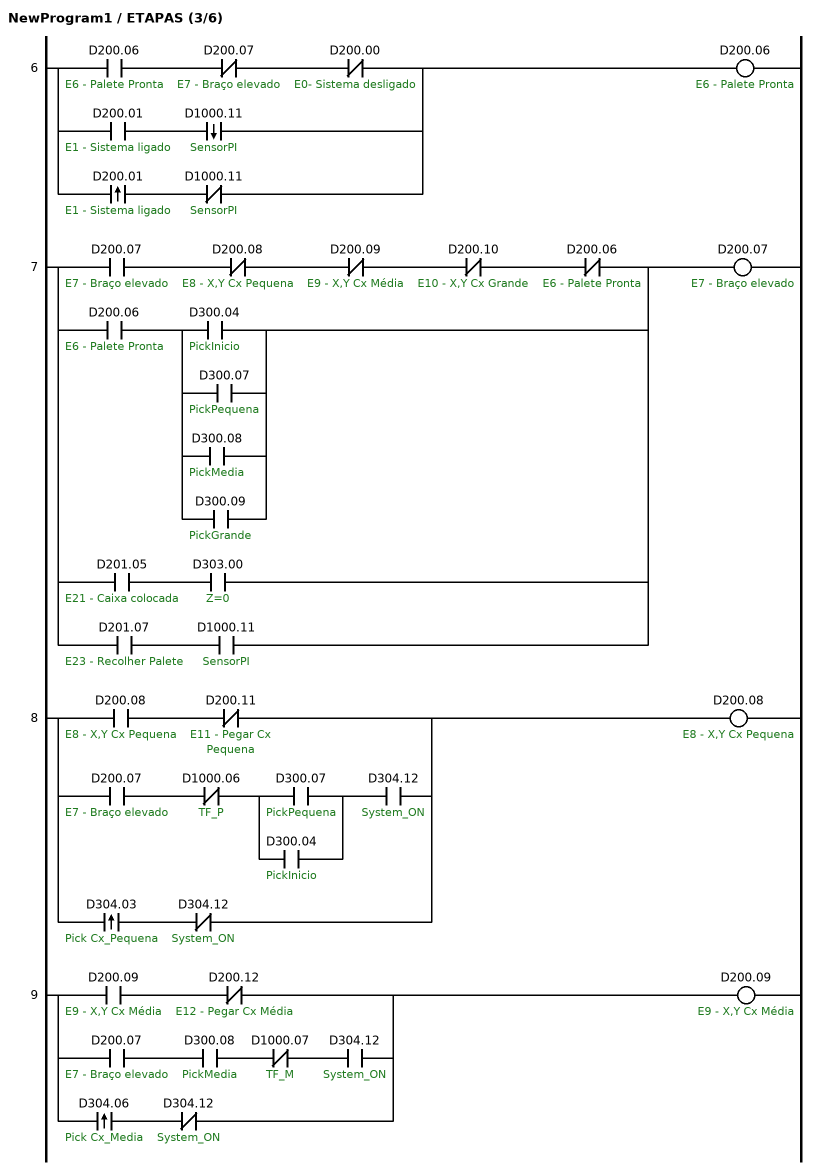
; rung 6
LD D200.06  ; E6 - Palete Pronta
ANDNOT D200.07  ; E7 - Braço elevado
ANDNOT D200.00  ; E0- Sistema desligado
LD D200.01  ; E1 - Sistema ligado
%AND D1000.11  ; SensorPI
ORLD
@LD D200.01  ; E1 - Sistema ligado
ANDNOT D1000.11  ; SensorPI
ORLD
OUT D200.06  ; E6 - Palete Pronta
; rung 7
LD D200.07  ; E7 - Braço elevado
ANDNOT D200.08  ; E8 - X,Y Cx Pequena
ANDNOT D200.09  ; E9 - X,Y Cx Média
ANDNOT D200.10  ; E10 - X,Y Cx Grande
ANDNOT D200.06  ; E6 - Palete Pronta
LD D200.06  ; E6 - Palete Pronta
LD D300.04  ; PickInicio
OR D300.07  ; PickPequena
OR D300.08  ; PickMedia
OR D300.09  ; PickGrande
ANDLD
ORLD
LD D201.05  ; E21 - Caixa colocada
AND D303.00  ; Z=0
ORLD
LD D201.07  ; E23 - Recolher Palete
AND D1000.11  ; SensorPI
ORLD
OUT D200.07  ; E7 - Braço elevado
; rung 8
LD D200.08  ; E8 - X,Y Cx Pequena
ANDNOT D200.11  ; E11 - Pegar Cx Pequena
LD D200.07  ; E7 - Braço elevado
ANDNOT D1000.06  ; TF_P
LD D300.07  ; PickPequena
OR D300.04  ; PickInicio
ANDLD
AND D304.12  ; System_ON
ORLD
@LD D304.03  ; Pick Cx_Pequena
ANDNOT D304.12  ; System_ON
ORLD
OUT D200.08  ; E8 - X,Y Cx Pequena
; rung 9
LD D200.09  ; E9 - X,Y Cx Média
ANDNOT D200.12  ; E12 - Pegar Cx Média
LD D200.07  ; E7 - Braço elevado
AND D300.08  ; PickMedia
ANDNOT D1000.07  ; TF_M
AND D304.12  ; System_ON
ORLD
@LD D304.06  ; Pick Cx_Media
ANDNOT D304.12  ; System_ON
ORLD
OUT D200.09  ; E9 - X,Y Cx Média

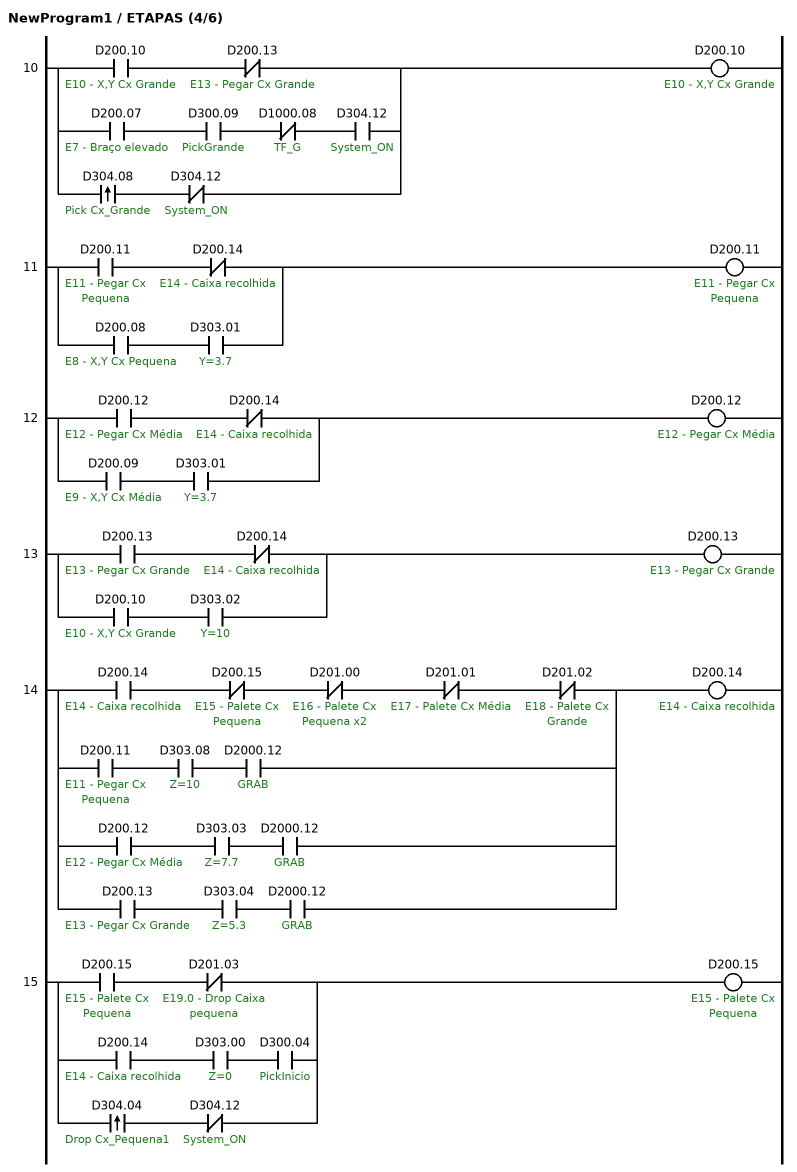
; rung 10
LD D200.10  ; E10 - X,Y Cx Grande
ANDNOT D200.13  ; E13 - Pegar Cx Grande
LD D200.07  ; E7 - Braço elevado
AND D300.09  ; PickGrande
ANDNOT D1000.08  ; TF_G
AND D304.12  ; System_ON
ORLD
@LD D304.08  ; Pick Cx_Grande
ANDNOT D304.12  ; System_ON
ORLD
OUT D200.10  ; E10 - X,Y Cx Grande
; rung 11
LD D200.11  ; E11 - Pegar Cx Pequena
ANDNOT D200.14  ; E14 - Caixa recolhida
LD D200.08  ; E8 - X,Y Cx Pequena
AND D303.01  ; Y=3.7
ORLD
OUT D200.11  ; E11 - Pegar Cx Pequena
; rung 12
LD D200.12  ; E12 - Pegar Cx Média
ANDNOT D200.14  ; E14 - Caixa recolhida
LD D200.09  ; E9 - X,Y Cx Média
AND D303.01  ; Y=3.7
ORLD
OUT D200.12  ; E12 - Pegar Cx Média
; rung 13
LD D200.13  ; E13 - Pegar Cx Grande
ANDNOT D200.14  ; E14 - Caixa recolhida
LD D200.10  ; E10 - X,Y Cx Grande
AND D303.02  ; Y=10
ORLD
OUT D200.13  ; E13 - Pegar Cx Grande
; rung 14
LD D200.14  ; E14 - Caixa recolhida
ANDNOT D200.15  ; E15 - Palete Cx Pequena
ANDNOT D201.00  ; E16 - Palete Cx Pequena x2
ANDNOT D201.01  ; E17 - Palete Cx Média
ANDNOT D201.02  ; E18 - Palete Cx Grande
LD D200.11  ; E11 - Pegar Cx Pequena
AND D303.08  ; Z=10
AND D2000.12  ; GRAB
ORLD
LD D200.12  ; E12 - Pegar Cx Média
AND D303.03  ; Z=7.7
AND D2000.12  ; GRAB
ORLD
LD D200.13  ; E13 - Pegar Cx Grande
AND D303.04  ; Z=5.3
AND D2000.12  ; GRAB
ORLD
OUT D200.14  ; E14 - Caixa recolhida
; rung 15
LD D200.15  ; E15 - Palete Cx Pequena
ANDNOT D201.03  ; E19.0 - Drop Caixa pequena
LD D200.14  ; E14 - Caixa recolhida
AND D303.00  ; Z=0
AND D300.04  ; PickInicio
ORLD
@LD D304.04  ; Drop Cx_Pequena1
ANDNOT D304.12  ; System_ON
ORLD
OUT D200.15  ; E15 - Palete Cx Pequena

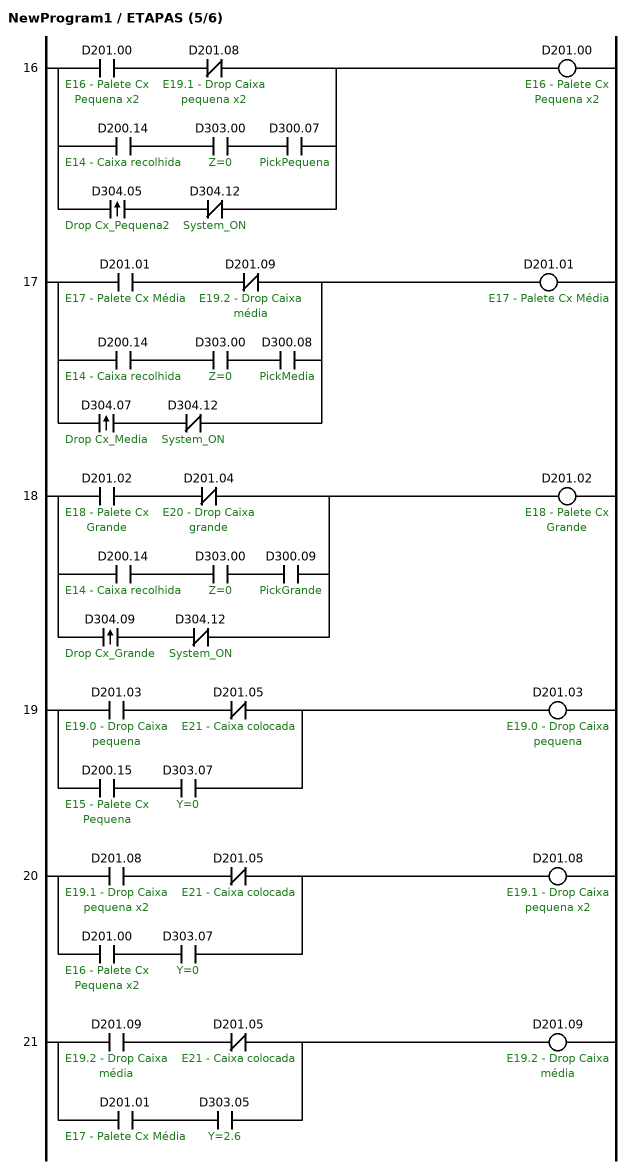
; rung 16
LD D201.00  ; E16 - Palete Cx Pequena x2
ANDNOT D201.08  ; E19.1 - Drop Caixa pequena x2
LD D200.14  ; E14 - Caixa recolhida
AND D303.00  ; Z=0
AND D300.07  ; PickPequena
ORLD
@LD D304.05  ; Drop Cx_Pequena2
ANDNOT D304.12  ; System_ON
ORLD
OUT D201.00  ; E16 - Palete Cx Pequena x2
; rung 17
LD D201.01  ; E17 - Palete Cx Média
ANDNOT D201.09  ; E19.2 - Drop Caixa média
LD D200.14  ; E14 - Caixa recolhida
AND D303.00  ; Z=0
AND D300.08  ; PickMedia
ORLD
@LD D304.07  ; Drop Cx_Media
ANDNOT D304.12  ; System_ON
ORLD
OUT D201.01  ; E17 - Palete Cx Média
; rung 18
LD D201.02  ; E18 - Palete Cx Grande
ANDNOT D201.04  ; E20 - Drop Caixa grande
LD D200.14  ; E14 - Caixa recolhida
AND D303.00  ; Z=0
AND D300.09  ; PickGrande
ORLD
@LD D304.09  ; Drop Cx_Grande
ANDNOT D304.12  ; System_ON
ORLD
OUT D201.02  ; E18 - Palete Cx Grande
; rung 19
LD D201.03  ; E19.0 - Drop Caixa pequena
ANDNOT D201.05  ; E21 - Caixa colocada
LD D200.15  ; E15 - Palete Cx Pequena
AND D303.07  ; Y=0
ORLD
OUT D201.03  ; E19.0 - Drop Caixa pequena
; rung 20
LD D201.08  ; E19.1 - Drop Caixa pequena x2
ANDNOT D201.05  ; E21 - Caixa colocada
LD D201.00  ; E16 - Palete Cx Pequena x2
AND D303.07  ; Y=0
ORLD
OUT D201.08  ; E19.1 - Drop Caixa pequena x2
; rung 21
LD D201.09  ; E19.2 - Drop Caixa média
ANDNOT D201.05  ; E21 - Caixa colocada
LD D201.01  ; E17 - Palete Cx Média
AND D303.05  ; Y=2.6
ORLD
OUT D201.09  ; E19.2 - Drop Caixa média

